INTERFACE ISimuMoverTimers

(* Process time, expressed in milisecond *)
PROPERTY iProcessTimeMili_1 : DINT
GET
END_GET
SET
END_SET
END_PROPERTY

(* Process time, expressed in milisecond *)
PROPERTY iProcessTimeMili_2 : DINT
GET
END_GET
SET
END_SET
END_PROPERTY

END_INTERFACE

(* stored: Version 1.1.0.1, ProductVersion 3.1.4024.6
   Itf ISimuMoverTimers: Id {3e53b767-d3d2-4389-aa58-689aee3700ca}
   Property iProcessTimeMili_1: Id {e14769f7-47e8-4324-ad81-884361f556c6}
   Get Get: Id {a404e07c-edad-4d45-b4f7-6097ec06d15c}
   Set Set: Id {222659ae-3b7c-400b-8d7f-dfbb06249b9e}
   Property iProcessTimeMili_2: Id {31e98800-1932-4e20-af14-e98484b89832}
   Get Get: Id {a8082181-d2b9-4efc-a70d-33c8c9c3e426}
   Set Set: Id {a1c93b54-4810-4ec4-b519-5c73fdefb6fb} *)
